Staubli VAL3: page_Production.dtx

mdesc mNomSpeed
bool bTrigger
bool bShowStatus
bool bMoveRelease
bool bLarge
bool bButton[8]
  [4] = true
  [5] = true
  [6] = true
  [7] = true
num nClockStatus
num nIndex
num nKey = -1
num nIndexItem
num nOldIndex
public num nPage
num nRefresh = 2164.601
num nSelected
num nTime = 1
num nType
num nView
pointRx pPointTest[7]
string sEvent = "hello"
string sEventImport
string sImport
public string sItems
string sList = "hello"
string sMenu[8]
  [0] = "Simulation"
  [4] = "Type"
  [5] = "Duplicate"
  [6] = "Delete"
  [7] = "New"
string sMenu8[8]
string sMenuUser[8]
string sMessage
string sTrsfNum[8 6]
string sWorkingmode[8]
